// When inherited, the child function block will gain two properties:
// InstanceName - ONLY the name of the instantiated function block
// InstancePath - the FULL instance path

{attribute 'reflection'}
{attribute 'hide_all_locals'}
{attribute 'no_explicit_call' := 'Body contains no logic, calling methods only allowed.'}
FUNCTION_BLOCK ABSTRACT FB_HasInstanceNameAndPath
VAR
	{attribute 'instance-path'} 
    {attribute 'noinit'} 
	_instancePath	: Tc2_System.T_MaxString;
	_instanceName	: Tc2_System.T_MaxString;
END_VAR

{attribute 'hide'}
METHOD FB_init : BOOL
VAR_INPUT
	bInitRetains : BOOL; // if TRUE, the retain variables are initialized (warm start / cold start)
	bInCopyCode : BOOL;  // if TRUE, the instance afterwards gets moved into the copy code (online change)
END_VAR
_instanceName := InstanceNameHelper.InstanceNameFromPath(_instancePath, 10);
_instancePath := InstanceNameHelper.RemoveProjectFromInstancePath(_instancePath);
END_METHOD

{attribute 'monitoring':='call'}
PROPERTY InstanceName : Tc2_System.T_MaxString
GET
InstanceName := _instanceName;
END_GET
END_PROPERTY

{attribute 'monitoring':='call'}
PROPERTY InstancePath : Tc2_System.T_MaxString
GET
VAR
	varInfo	: T_VarInfo;
END_VAR
InstancePath := _instancePath;
END_GET
END_PROPERTY

END_FUNCTION_BLOCK

(* stored: Version 1.1.0.1, ProductVersion 3.1.4024.14
   POU FB_HasInstanceNameAndPath: Id {87d42491-7a36-0b06-1027-fbe6e5b19dcf}, SpecialFunc None
   Method FB_init: Id {b1ecb943-9b1e-0f5b-3348-047bf079c662}
   Property InstanceName: Id {0894143d-927f-0465-344c-14f9b9c738ea}
   Get Get: Id {b959f917-9381-0887-27aa-c909d33f58f6}
   Property InstancePath: Id {9665f2f7-723f-06f2-2fd9-4941869795b6}
   Get Get: Id {280f29c4-2287-0abd-1386-09c1556898dc} *)
